Yaskawa INFORM job: X2_100(P)(125,-90).JBI

/JOB
//NAME X2_100(P)(125,-90)
//POS
///NPOS 391,391,391,27,0,0
///TOOL 0
///POSTYPE PULSE
///PULSE
C00000=15474,202180,164610,0,0,38
C00001=2027,202198,164679,0,0,38
C00002=24736,215365,219614,34446,41710,-28276
C00003=32352,212431,219590,43411,47182,-30672
C00004=90146,188560,202920,30112,59119,-18336
C00005=118933,140461,218744,27304,53624,2807
C00006=119754,138493,231524,24113,52403,6590
C00007=120507,123084,224138,21975,53379,9268
C00008=120855,115436,217153,22091,53699,9378
C00009=120999,112276,214168,22121,53888,9436
C00010=120994,108702,209954,21918,54592,9592
C00011=121002,109206,210530,21948,54503,9573
C00012=121014,109176,212154,22227,53559,9363
C00013=121002,109206,210530,21948,54503,9573
C00014=120510,120230,220891,21834,53874,9379
C00015=120545,123144,224216,-26507,40921,-26256
C00016=120895,115499,217236,-26128,41279,-26328
C00017=121036,110360,211926,-25743,41856,-26497
C00018=121034,108769,210044,-25582,42165,-26596
C00019=121035,109319,210673,-25631,42070,-26566
C00020=121049,109287,212294,-26118,41154,-26266
C00021=121035,109319,210673,-25631,42070,-26566
C00022=120543,120334,221019,-26244,41392,-26415
C00023=120983,122786,223558,-30476,46746,-26242
C00024=120987,115437,217242,-30421,46842,-26276
C00025=120987,110819,212678,-30218,47221,-26411
C00026=120984,108845,210344,-30028,47588,-26540
C00027=121056,109448,211035,-30038,47494,-26498
C00028=121070,109406,212645,-30499,46616,-26184
C00029=121056,109448,211035,-30038,47494,-26498
C00030=121048,120014,220398,-30195,47204,-26397
C00031=120925,149751,244690,-34380,46703,-25518
C00032=121565,167094,227706,-36094,61868,-28983
C00033=121107,161331,224195,-36551,61107,-28820
C00034=120919,157058,220850,-36681,60950,-28811
C00035=120917,155800,219633,-36648,61033,-28842
C00036=120923,156278,220067,-36652,61017,-28835
C00037=120930,157317,222816,-37031,60082,-28475
C00038=120923,156278,220067,-36652,61017,-28835
C00039=121567,164501,225300,-36048,61989,-29027
C00040=120589,166944,227359,-19824,59976,-30928
C00041=120819,161134,223823,-19888,59243,-30737
C00042=120912,157183,220866,-19892,59057,-30681
C00043=120909,155576,219240,-19859,59222,-30713
C00044=120921,156089,219731,-19862,59188,-30703
C00045=120928,157137,222490,-20094,58096,-30494
C00046=120921,156089,219731,-19862,59188,-30703
C00047=120597,164381,225001,-19795,60104,-30950
C00048=133714,167013,227584,29806,67145,20919
C00049=134110,161138,223906,30151,66407,20805
C00050=134262,157498,221144,30262,66227,20790
C00051=134252,155557,219269,30222,66366,20826
C00052=134278,156050,219725,30241,66337,20824
C00053=134486,157077,222435,30590,65306,20576
C00054=134278,156050,219725,30241,66337,20824
C00055=133722,164435,225200,29782,67268,20955
C00056=133985,188744,240463,29202,55916,39414
C00057=133788,188005,227705,27049,47808,60336
C00058=134139,183273,225821,27621,46590,60080
C00059=134274,179997,223870,27848,46130,59979
C00060=134264,178443,222562,27844,46137,59979
C00061=134276,178874,222921,27846,46135,59983
C00062=134459,180391,226047,28389,45077,59697
C00063=134276,178874,222921,27846,46135,59983
C00064=133784,185635,225817,27071,47759,60319
C00065=127585,202169,243145,858,47044,1942
C00066=121193,187855,227430,-25535,51149,-56270
C00067=120989,183220,225717,-26035,49903,-55992
C00068=120906,180048,223892,-26233,49429,-55882
C00069=120903,178425,222522,-26231,49435,-55886
C00070=120895,178865,222881,-26231,49438,-55890
C00071=120901,180413,226062,-26675,48393,-55581
C00072=120895,178865,222881,-26231,49438,-55890
C00073=121182,185490,225532,-25553,51104,-56261
C00074=121188,188192,227969,-25590,51004,-56232
C00075=120983,183552,226258,-26095,49755,-55951
C00076=120899,180084,224188,-26297,49279,-55843
C00077=120898,178760,223074,-26295,49283,-55844
C00078=120902,179187,223391,-26285,49306,-55850
C00079=120908,180723,226556,-26731,48265,-55540
C00080=120902,179187,223391,-26285,49306,-55850
C00081=121189,185816,226036,-25601,50976,-56224
C00082=123255,190499,236374,-58349,45147,30432
C00083=121547,184669,229695,-57916,45057,29536
C00084=120879,180825,225690,-57693,45050,29154
C00085=120877,179386,224486,-57692,45050,29153
C00086=120865,179866,224825,-57664,45066,29131
C00087=120860,178282,221599,-56698,45720,28507
C00088=120865,179866,224825,-57664,45066,29131
C00089=120725,179892,223679,-57103,45408,28721
C00090=120332,179896,223682,-57208,45243,28650
C00091=121348,179880,223660,-56933,45672,28832
C00092=123711,188247,233364,-57633,45714,30138
C00093=134983,214876,238244,-8707,44220,8832
C00094=134548,207430,231310,-8578,44619,8625
C00095=134367,202745,227274,-8541,44679,8550
C00096=134362,201870,226673,-8552,44600,8555
C00097=134379,202451,227139,-8553,44612,8561
C00098=134212,200435,223640,-8367,45704,8394
C00099=134379,202451,227139,-8553,44612,8561
C00100=134984,213013,237167,-8753,43928,8861
C00101=144264,210294,243886,-8163,41086,13861
C00102=162452,180370,234066,-6629,37835,23828
C00103=161533,173092,227071,-6569,38350,23478
C00104=162432,167522,220632,-6394,39487,23686
C00105=162432,166208,219497,-6392,39511,23685
C00106=162432,166481,219733,-6392,39506,23685
C00107=161891,165056,216873,-6255,40502,23429
C00108=162432,166481,219733,-6392,39506,23685
C00109=162497,178365,232600,-6647,37710,23854
C00110=147308,180890,237204,47154,21007,-10994
C00111=147638,173377,228129,43966,22135,-9369
C00112=147769,169207,223427,42684,22650,-8713
C00113=147776,167383,221906,42683,22648,-8711
C00114=147797,168129,222540,42691,22636,-8708
C00115=147426,166532,219395,41033,23590,-8010
C00116=147797,168129,222540,42691,22636,-8708
C00117=147340,178856,235656,47326,20933,-11067
C00118=133884,161941,227787,33603,50676,10210
C00119=127576,130559,218004,30921,63820,21625
C00120=128836,119462,220153,33793,57797,19920
C00121=129449,112387,214292,34197,57712,19962
C00122=129575,109480,211887,34296,57687,19970
C00123=132342,109409,211410,35968,57614,20273
C00124=135809,109300,210711,38054,57534,20678
C00125=138378,109197,210091,39570,57490,20998
C00126=138013,112115,212550,39343,57524,20963
C00127=137185,119214,218524,38825,57601,20885
C00128=115991,118707,218017,-25490,47827,-39243
C00129=116216,112084,213018,-25487,47549,-39133
C00130=116067,109362,210943,-25621,47425,-39117
C00131=124525,109336,210994,-20745,47997,-38204
C00132=124884,112043,212960,-20482,48190,-38202
C00133=124386,118675,218008,-20675,48440,-38320
C00134=123290,120759,219660,-35956,60120,-26268
C00135=122628,114303,214891,-36511,59734,-26205
C00136=121471,111489,212711,-37298,59521,-26266
C00137=122737,102232,205148,-46823,63858,-23746
C00138=124301,104933,207355,-45758,64087,-23652
C00139=125674,111471,212543,-44779,64387,-23617
C00140=122699,156385,234573,-36508,60394,-36922
C00141=122451,163606,222345,-33636,69881,-40152
C00142=121996,159570,221367,-34155,68543,-39836
C00143=121756,157914,220964,-34404,67985,-39712
C00144=120095,157879,220889,-35223,67629,-40000
C00145=118379,157761,220797,-36072,67224,-40285
C00146=122498,151785,218689,-44973,69197,-37741
C00147=123062,153607,219376,-44540,69722,-37837
C00148=123990,157704,220658,-43734,70938,-38144
C00149=117621,162254,221874,-19766,66589,-43069
C00150=117804,158098,220771,-19895,65240,-42790
C00151=117692,155503,219422,-20025,64751,-42727
C00152=123564,155493,219421,-17329,65494,-41580
C00153=123448,158048,220704,-17317,65981,-41679
C00154=123147,162227,221856,-17278,67320,-41949
C00155=130667,163848,224751,30344,74631,25358
C00156=131102,158990,222619,30735,73515,25150
C00157=131194,156955,221592,30843,73138,25067
C00158=136997,155740,218820,33776,72826,26305
C00159=136728,157787,219942,33579,73190,26353
C00160=136199,162650,222153,33133,74269,26558
C00161=131924,177838,230931,28709,51404,58848
C00162=131093,185219,225656,26178,57978,60553
C00163=131486,181652,225386,26742,56390,60255
C00164=131623,179818,224816,26950,55830,60146
C00165=136523,178332,222014,27857,55574,61608
C00166=136419,180039,222404,27637,56164,61742
C00167=135955,197166,232402,26774,58642,62268
C00168=123486,183195,222462,-21671,66302,-58170
C00169=123320,180439,223276,-22038,64485,-57858
C00170=123006,178865,223348,-22286,63635,-57774
C00171=118045,178731,223219,-23875,62688,-58963
C00172=118318,180513,223383,-23631,63488,-59060
C00173=118578,183298,222619,-23202,65292,-59373
C00174=122208,184099,222550,-27312,66798,-58279
C00175=121800,181437,223437,-27825,64995,-57938
C00176=121432,179848,223509,-28133,64143,-57821
C00177=118640,179803,223425,-29053,63504,-58468
C00178=122362,176158,223733,-39099,63902,-56258
C00179=122919,177928,223953,-38663,64680,-56393
C00180=123741,180697,223374,-37873,66345,-56772
C00181=125859,202099,241745,-26899,43318,-21165
C00182=128113,178960,235420,-24516,16567,13756
C00183=127689,171451,226207,-21929,18167,12428
C00184=127528,167831,221933,-20974,18864,11937
C00185=125917,168120,222387,-19991,18484,11020
C00186=112964,167943,221792,-9276,17273,2399
C00187=116391,165192,218668,-37133,21773,16827
C00188=116794,168607,222919,-38620,21196,17655
C00189=117426,176109,232276,-42123,19905,19505
C00190=121934,189549,236157,-2154,24440,9441
C00191=125766,180591,223933,31743,27648,1072
C00192=125872,172130,214005,30040,29143,1966
C00193=126601,167752,208377,28765,30022,2815
C00194=142051,161046,196707,20020,29981,11317
C00195=142147,165297,201916,20601,29000,11042
C00196=142364,174552,213002,21900,27026,10440
C00197=90146,188560,202920,30112,59119,-18336
C00198=32352,212431,219590,43411,47182,-30672
C00199=2027,202198,164679,0,0,38
C00200=15474,202180,164610,0,0,38
C00201=15474,202180,164610,0,0,38
C00202=15474,202180,164610,0,0,38
C00203=15474,202180,164610,0,0,38
C00204=15474,202180,164610,0,0,38
C00205=-58614,195716,224396,-17895,28031,-14924
C00206=-117113,152285,229609,-38431,39797,-17389
C00207=-135921,136983,237719,-46639,40267,-16819
C00208=-146165,113701,216007,-48123,45886,-19082
C00209=-147115,109767,211721,-48018,46725,-19481
C00210=-147088,107791,209384,-47709,47018,-19672
C00211=-147094,108297,209962,-47779,46951,-19629
C00212=-147691,108253,211472,-48816,46225,-19236
C00213=-147094,108297,209962,-47779,46951,-19629
C00214=-145940,119401,220708,-47691,46482,-19124
C00215=-145956,122257,223946,12736,42114,23473
C00216=-146776,114562,216701,12165,42638,23451
C00217=-149521,110157,218004,11318,39720,22735
C00218=-147064,107789,209368,11782,43659,23556
C00219=-152611,108638,222377,10271,36372,22002
C00220=-147661,108297,211513,11684,42643,23344
C00221=-152611,108638,222377,10271,36372,22002
C00222=-145911,119443,220742,12635,42626,23555
C00223=-129100,127332,227576,23440,42260,25369
C00224=-99845,140323,234668,41114,43975,29200
C00225=-81288,119441,205391,47500,48209,34399
C00226=-80509,111680,198241,47632,48326,34680
C00227=-79929,105264,191953,47555,48593,35008
C00228=-79929,103140,189447,47268,48904,35206
C00229=-79929,103522,189901,47320,48847,35170
C00230=-79411,103879,191333,48035,48251,34928
C00231=-80657,107851,193513,46953,49010,35078
C00232=-81393,116289,201791,47062,48643,34649
C00233=-121441,148548,228494,40235,53726,25728
C00234=-121126,165586,226218,36457,61785,29251
C00235=-120656,159787,222623,36910,61050,29098
C00236=-120465,155988,219703,37047,60878,29083
C00237=-120464,154211,217972,36998,61001,29130
C00238=-120470,154693,218414,37003,60983,29122
C00239=-120461,155760,221201,37395,60041,28759
C00240=-120470,154693,218414,37003,60983,29122
C00241=-121130,162973,223775,36406,61917,29299
C00242=-120157,165759,226450,20196,59859,31167
C00243=-120376,159925,222865,20264,59145,30979
C00244=-120465,156088,219927,20262,59004,30931
C00245=-120464,154338,218223,20232,59143,30959
C00246=-120475,154854,218720,20235,59107,30949
C00247=-120466,155913,221497,20480,58011,30738
C00248=-120475,154854,218720,20235,59107,30949
C00249=-120168,163183,224065,20164,59996,31190
C00250=-146488,166005,227001,-35633,64430,-23031
C00251=-147030,160017,223073,-36069,63762,-22930
C00252=-147236,156149,220027,-36198,63621,-22931
C00253=-147219,154376,218307,-36149,63745,-22972
C00254=-147245,154867,218758,-36168,63719,-22970
C00255=-147633,155852,221361,-36670,62738,-22707
C00256=-147245,154867,218758,-36168,63719,-22970
C00257=-146483,163417,224595,-35590,64555,-23074
C00258=-120317,171933,242187,-34338,35763,-50845
C00259=-120155,165766,226473,-29925,41593,-53256
C00260=-120374,159929,222883,-30422,40861,-53041
C00261=-120463,156296,220142,-30547,40687,-53000
C00262=-120462,154340,218238,-30449,40831,-53058
C00263=-120473,154616,218516,-30468,40803,-53050
C00264=-120468,155465,220597,-30969,40075,-52744
C00265=-120473,154822,218708,-30475,40793,-53046
C00266=-120165,163158,224064,-29848,41715,-53306
C00267=-120812,165753,226464,30411,41431,53453
C00268=-120571,159914,222865,30920,40700,53240
C00269=-120472,156279,220119,31048,40527,53200
C00270=-120471,154323,218216,30948,40670,53260
C00271=-120462,154817,218686,30971,40637,53250
C00272=-120453,155874,221461,31687,39633,52832
C00273=-120462,154817,218686,30971,40637,53250
C00274=-120802,163155,224052,30328,41558,53507
C00275=-120794,196445,225743,23944,55971,57861
C00276=-120590,192435,224899,24399,54512,57575
C00277=-120507,189535,223519,24597,53909,57452
C00278=-120506,188039,222351,24612,53862,57441
C00279=-120510,188436,222616,24600,53901,57449
C00280=-120503,190244,226011,24956,52841,57180
C00281=-120510,188436,222616,24600,53901,57449
C00282=-120797,194186,224030,23972,55873,57836
C00283=-120994,201212,234683,5149,48132,-3005
C00284=-136826,197795,228776,4624,50735,-8156
C00285=-136826,191727,224657,4661,50153,-8183
C00286=-138745,198654,246113,16555,26136,-13965
C00287=-138745,196808,244858,16658,25967,-14016
C00288=-138745,198654,246113,16555,26136,-13965
C00289=-138556,197554,243943,16057,26850,-13661
C00290=-138745,198654,246113,16555,26136,-13965
C00291=-120778,201953,235347,5155,48094,-2935
C00292=-122925,194375,228384,5084,48585,-3628
C00293=-122022,191255,226196,5106,48287,-3341
C00294=-122022,188924,224535,5119,48113,-3349
C00295=-122022,191255,226196,5106,48287,-3341
C00296=-122007,189355,222871,5025,49352,-3280
C00297=-122022,191255,226196,5106,48287,-3341
C00298=-120785,199939,233992,5171,47894,-2948
C00299=-121100,206663,244168,5684,44070,-5780
C00300=-121083,191157,235435,5956,40419,-9249
C00301=-120661,183492,227908,5865,41088,-9055
C00302=-120495,180342,224726,5822,41418,-8974
C00303=-120493,177643,222664,5836,41300,-8982
C00304=-120497,178404,223351,5840,41268,-8985
C00305=-120504,176471,219821,5709,42442,-8908
C00306=-120497,178404,223351,5840,41268,-8985
C00307=-121086,189297,234244,5983,40198,-9266
C00308=-146820,179847,236540,-47569,21348,11498
C00309=-147178,172319,227421,-44381,22472,9861
C00310=-147319,168316,222840,-43092,22988,9195
C00311=-147327,166302,221149,-43081,22990,9188
C00312=-147348,167051,221792,-43093,22976,9188
C00313=-146991,165439,218615,-41422,23930,8479
C00314=-147348,167051,221792,-43093,22976,9188
C00315=-146852,177807,234978,-47728,21278,11565
C00316=-135233,175637,232065,-30395,22918,7865
C00317=-134932,170558,225163,-28644,24419,7102
C00318=-134048,167164,221268,-28229,25184,7160
C00319=-151719,157645,202807,-16034,27960,-3795
C00320=-149884,166658,215825,-18859,24998,-1880
C00321=-146998,184619,240811,-25863,19770,2323
C00322=-125978,166364,224291,9417,26840,-6325
C00323=-129674,155803,216839,10617,26282,-8064
C00324=-129498,149917,208752,9902,28190,-7650
C00325=-128727,145711,203487,9397,29196,-7156
C00326=-146983,136453,186134,10957,36521,-13611
C00327=-147815,150895,204985,12306,32503,-14599
C00328=-147815,166494,219236,12563,31767,-14734
C00329=-117911,183214,223223,-22567,61413,-57159
C00330=-118075,179761,223119,-22973,59798,-56859
C00331=-118640,177544,221909,-23214,59324,-56920
C00332=-123472,177522,221869,-24524,58369,-58124
C00333=-123089,179795,223206,-24339,58762,-58103
C00334=-122842,183276,223359,-23878,60366,-58401
C00335=-123442,190112,227842,21784,66477,58404
C00336=-123264,179517,222829,22229,64249,58012
C00337=-123470,177948,222872,22311,63517,57806
C00338=-118464,178077,223118,23939,62475,58981
C00339=-118255,179504,222781,23818,63292,59223
C00340=-118526,182312,222057,23382,65085,59534
C00341=-122160,182951,221704,27481,66647,58451
C00342=-121741,180270,222553,28000,64855,58113
C00343=-121841,178346,222179,28131,64207,57913
C00344=-118577,178303,222154,29213,63422,58659
C00345=-122472,175017,222795,39229,63796,56395
C00346=-122854,176802,223069,38864,64502,56556
C00347=-123688,179595,222537,38068,66154,56931
C00348=-122762,177463,230138,35132,68647,45006
C00349=-122410,162609,221657,33920,69712,40281
C00350=-121942,158550,220632,34447,68388,39967
C00351=-122084,156654,219964,34496,67953,39787
C00352=-118316,156835,220042,36358,67113,40432
C00353=-122608,150908,218064,45207,69057,37831
C00354=-122995,152587,218620,44867,69536,37955
C00355=-123937,156712,219961,44053,70736,38256
C00356=-117567,161316,221321,20040,66440,43208
C00357=-117737,157140,220183,20178,65102,42929
C00358=-118356,154594,218971,19982,64654,42713
C00359=-123958,154557,218888,17402,65396,41629
C00360=-123397,157158,220257,17595,65803,41812
C00361=-123107,161358,221443,17548,67132,42081
C00362=-143812,163767,225728,-37102,71366,-27286
C00363=-144478,158774,223325,-37668,70333,-27076
C00364=-145574,156483,221747,-38290,69906,-27183
C00365=-150790,154198,216554,-40571,70164,-28612
C00366=-149872,156514,218237,-40068,70526,-28516
C00367=-149135,161509,220758,-39481,71513,-28708
C00368=-132073,148583,237547,-34621,60846,-21391
C00369=-128841,120799,222047,-33572,57550,-19735
C00370=-130509,111569,213679,-34507,57728,-19991
C00371=-142163,108136,208271,-41379,57632,-21462
C00372=-150058,107393,204742,-45605,57822,-22784
C00373=-138074,111342,212170,-39066,57558,-20867
C00374=-137251,118465,218184,-38555,57622,-20786
C00375=-115920,117937,217688,25888,47668,39306
C00376=-117242,111297,212709,25258,47458,39075
C00377=-117220,108280,210223,25280,47439,39073
C00378=-125843,108493,210262,20260,48127,38171
C00379=-124861,111270,212684,20846,48005,38264
C00380=-124377,117927,217775,21034,48243,38378
C00381=-123273,119993,219247,36349,59987,26322
C00382=-122589,113511,214424,36914,59617,26265
C00383=-122996,110841,212352,36684,59583,26203
C00384=-117053,110850,212325,40539,58921,26676
C00385=-124086,101367,204591,46303,63921,23704
C00386=-124243,104084,206817,46189,63960,23705
C00387=-125643,110657,212075,45198,64245,23661
C00388=-113480,133194,224663,34991,55578,15993
C00389=-58614,195716,224396,-17895,28031,-14924
C00390=15474,202180,164610,0,0,38
BC00000=0,675528,1075229
BC00001=0,1249520,1075229
BC00002=20074,1273230,1075229
BC00003=22843,1276500,1075229
BC00004=181219,1349640,881743
BC00005=259614,1271622,997019
BC00006=263455,1253369,961473
BC00007=265649,1242939,941161
BC00008=265649,1242939,941161
BC00009=265649,1242939,941161
BC00010=265649,1242939,941161
BC00011=265649,1242939,941161
BC00012=265649,1242939,941161
BC00013=265649,1242939,941161
BC00014=265649,1242939,941161
BC00015=279094,1259762,979345
BC00016=279094,1259762,979345
BC00017=279094,1259762,979345
BC00018=279094,1259762,979345
BC00019=279094,1259762,979345
BC00020=279094,1259762,979345
BC00021=279094,1259762,979345
BC00022=279094,1259762,979345
BC00023=338482,1253298,958814
BC00024=338482,1253298,958814
BC00025=338482,1253298,958814
BC00026=338482,1253298,958814
BC00027=338482,1253298,958814
BC00028=338482,1253298,958814
BC00029=338482,1253298,958814
BC00030=338482,1253298,958814
BC00031=333821,1266832,919202
BC00032=321005,1304050,810268
BC00033=321005,1304050,810268
BC00034=321005,1304050,810268
BC00035=321005,1304050,810268
BC00036=321005,1304050,810268
BC00037=321005,1304050,810268
BC00038=321005,1304050,810268
BC00039=321005,1304050,810268
BC00040=279090,1297669,836196
BC00041=279090,1297669,836196
BC00042=279090,1297669,836196
BC00043=279090,1297669,836196
BC00044=279090,1297669,836196
BC00045=279090,1297669,836196
BC00046=279090,1297669,836196
BC00047=279090,1297669,836196
BC00048=308990,1283728,803935
BC00049=308990,1283728,803935
BC00050=308990,1283728,803935
BC00051=308990,1283728,803935
BC00052=308990,1283728,803935
BC00053=308990,1283728,803935
BC00054=308990,1283728,803935
BC00055=308990,1283728,803935
BC00056=309388,1296619,799441
BC00057=309813,1310369,794648
BC00058=309813,1310369,794648
BC00059=309813,1310369,794648
BC00060=309813,1310369,794648
BC00061=309813,1310369,794648
BC00062=309813,1310369,794648
BC00063=309813,1310369,794648
BC00064=309813,1310369,794648
BC00065=290509,1311906,794287
BC00066=271204,1313444,793926
BC00067=271204,1313444,793926
BC00068=271204,1313444,793925
BC00069=271204,1313444,793926
BC00070=271204,1313444,793926
BC00071=271204,1313444,793926
BC00072=271204,1313444,793926
BC00073=271204,1313444,793926
BC00074=339752,1313535,794120
BC00075=339752,1313535,794120
BC00076=339752,1313535,794120
BC00077=339752,1313535,794120
BC00078=339752,1313535,794120
BC00079=339752,1313535,794120
BC00080=339752,1313535,794120
BC00081=339752,1313535,794120
BC00082=309596,1336055,723788
BC00083=309596,1336055,723788
BC00084=309596,1336055,723788
BC00085=309596,1336055,723788
BC00086=309596,1336055,723788
BC00087=309596,1336055,723788
BC00088=309596,1336055,723788
BC00089=309596,1336055,723788
BC00090=309596,1336055,723788
BC00091=309596,1336055,723788
BC00092=309596,1336055,723788
BC00093=366840,1349942,659049
BC00094=366840,1349942,659049
BC00095=366840,1349942,659049
BC00096=366840,1349942,659049
BC00097=366840,1349942,659049
BC00098=366840,1349942,659049
BC00099=366840,1349942,659049
BC00100=366840,1349942,659049
BC00101=369598,1321086,746352
BC00102=375224,1262220,924452
BC00103=375224,1262220,924452
BC00104=375224,1262220,924452
BC00105=375224,1262220,924452
BC00106=375224,1262220,924452
BC00107=375224,1262220,924450
BC00108=375224,1262220,924452
BC00109=375224,1262220,924452
BC00110=339925,1300732,881743
BC00111=339925,1300732,881743
BC00112=339925,1300732,881743
BC00113=339925,1300732,881743
BC00114=339925,1300732,881743
BC00115=339925,1300732,881743
BC00116=339925,1300732,881743
BC00117=339925,1300732,881743
BC00118=315652,1292340,901479
BC00119=299654,1262212,953023
BC00120=298993,1238691,912276
BC00121=298993,1238691,912276
BC00122=298993,1238691,912274
BC00123=298993,1238691,912276
BC00124=298993,1238691,912276
BC00125=298993,1238691,912276
BC00126=298993,1238691,912276
BC00127=298993,1238691,912276
BC00128=278815,1248832,951478
BC00129=278815,1248832,951478
BC00130=278815,1248832,951478
BC00131=278815,1248832,951478
BC00132=278815,1248832,951478
BC00133=278815,1248832,951478
BC00134=314804,1246682,892728
BC00135=314804,1246682,892728
BC00136=314804,1246682,892728
BC00137=314804,1246682,892728
BC00138=314804,1246682,892728
BC00139=314804,1246682,892728
BC00140=314801,1292959,892910
BC00141=314719,1294052,772836
BC00142=314719,1294052,772836
BC00143=314719,1294052,772836
BC00144=314719,1294052,772836
BC00145=314719,1294052,772836
BC00146=314719,1294052,772836
BC00147=314719,1294052,772836
BC00148=314719,1294052,772836
BC00149=278878,1286739,810029
BC00150=278878,1286739,810029
BC00151=278878,1286739,810029
BC00152=278878,1286739,810029
BC00153=278878,1286739,810029
BC00154=278878,1286739,810029
BC00155=311908,1275469,768683
BC00156=311908,1275469,768683
BC00157=311908,1275469,768683
BC00158=311908,1275469,768683
BC00159=311908,1275469,768683
BC00160=311908,1275469,768683
BC00161=311248,1293583,920117
BC00162=310634,1294320,778613
BC00163=310634,1294320,778613
BC00164=310635,1294320,778611
BC00165=310635,1294320,778611
BC00166=310634,1294320,778613
BC00167=310634,1294320,778613
BC00168=269571,1288878,766650
BC00169=269571,1288878,766650
BC00170=269571,1288878,766650
BC00171=269571,1288878,766650
BC00172=269571,1288878,766650
BC00173=269571,1288878,766650
BC00174=324029,1292263,751538
BC00175=324029,1292263,751538
BC00176=324029,1292263,751538
BC00177=324029,1292263,751538
BC00178=324029,1292263,751538
BC00179=324029,1292263,751538
BC00180=324029,1292263,751538
BC00181=331457,1324273,767907
BC00182=337552,1339765,848258
BC00183=337552,1339765,848258
BC00184=337551,1339764,848257
BC00185=337552,1339765,848258
BC00186=337552,1339765,848258
BC00187=337552,1339765,848258
BC00188=337552,1339765,848258
BC00189=337552,1339765,848258
BC00190=326395,1340304,844891
BC00191=315775,1339017,839253
BC00192=315775,1339017,839253
BC00193=315775,1339017,839253
BC00194=315775,1339017,839253
BC00195=315775,1339017,839253
BC00196=315775,1339017,839253
BC00197=181219,1349640,881743
BC00198=22843,1276500,1075229
BC00199=0,1249520,1075229
BC00200=0,675528,1075229
BC00201=0,675528,1075229
BC00202=0,675528,1075229
BC00203=0,675528,1075229
BC00204=0,675528,1075229
BC00205=138607,763027,1056836
BC00206=261748,840763,986656
BC00207=303122,866882,963076
BC00208=320914,878114,952936
BC00209=322510,879121,952026
BC00210=322510,879121,952026
BC00211=322510,879121,952026
BC00212=322510,879121,952026
BC00213=322510,879121,952026
BC00214=322510,879121,952026
BC00215=326477,871688,980713
BC00216=326477,871688,980713
BC00217=326477,883252,980713
BC00218=326477,871688,980713
BC00219=326477,895644,980713
BC00220=326477,871688,980713
BC00221=326477,895644,980713
BC00222=326477,871688,980713
BC00223=304746,865718,972507
BC00224=267497,855485,958441
BC00225=255081,864777,953752
BC00226=255081,864777,953752
BC00227=255081,864777,953752
BC00228=255081,864777,953752
BC00229=255081,864777,953752
BC00230=255081,864777,953752
BC00231=255081,864777,953752
BC00232=255081,864777,953752
BC00233=320924,819371,961652
BC00234=320924,819371,812233
BC00235=320924,819371,812233
BC00236=320924,819371,812233
BC00237=320924,819371,812233
BC00238=320924,819371,812233
BC00239=320924,819371,812233
BC00240=320924,819371,812233
BC00241=320924,819371,812233
BC00242=278908,825639,838037
BC00243=278908,825639,838037
BC00244=278908,825639,838037
BC00245=278908,825639,838037
BC00246=278908,825639,838037
BC00247=278908,825639,838037
BC00248=278908,825639,838037
BC00249=278908,825639,838037
BC00250=344258,850073,804397
BC00251=344258,850073,804397
BC00252=344258,850073,804397
BC00253=344258,850073,804397
BC00254=344258,850073,804397
BC00255=344258,850073,804397
BC00256=344258,850073,804397
BC00257=344258,850073,804397
BC00258=268540,837164,928608
BC00259=268540,837164,928608
BC00260=268540,837164,928608
BC00261=268540,837164,928608
BC00262=268540,837164,928608
BC00263=268540,837164,928608
BC00264=268541,837164,928607
BC00265=268540,837164,928608
BC00266=268540,837164,928608
BC00267=271645,836699,929417
BC00268=271645,836699,929417
BC00269=271645,836699,929417
BC00270=271645,836699,929417
BC00271=271645,836699,929417
BC00272=271645,836699,929417
BC00273=271645,836699,929417
BC00274=271645,836699,929417
BC00275=340192,799254,723936
BC00276=340192,799254,723936
BC00277=340192,799254,723936
BC00278=340192,799254,723936
BC00279=340192,799254,723936
BC00280=340192,799254,723936
BC00281=340192,799254,723936
BC00282=340192,799254,723936
BC00283=321646,797982,745635
BC00284=321646,797982,745635
BC00285=321646,797982,745635
BC00286=321646,797982,745635
BC00287=321646,797982,745635
BC00288=321646,797982,745635
BC00289=321646,797982,745635
BC00290=321646,797982,745635
BC00291=321646,797982,745635
BC00292=321646,797982,745635
BC00293=321646,797984,745632
BC00294=321646,797984,745632
BC00295=321646,797984,745632
BC00296=321646,797984,745632
BC00297=321646,797984,745632
BC00298=321646,797982,745635
BC00299=296475,807012,791430
BC00300=260705,819844,856508
BC00301=260705,819844,856508
BC00302=260705,819844,856508
BC00303=260705,819844,856508
BC00304=260705,819844,856508
BC00305=260705,819844,856508
BC00306=260705,819844,856508
BC00307=260705,819844,856508
BC00308=339123,823007,883432
BC00309=339123,823007,883432
BC00310=339123,823007,883432
BC00311=339123,823007,883432
BC00312=339123,823007,883432
BC00313=339123,823007,883432
BC00314=339123,823007,883432
BC00315=339123,823007,883432
BC00316=339668,815369,895136
BC00317=339668,815369,895136
BC00318=339668,815369,895136
BC00319=339682,815172,895438
BC00320=339682,815172,895438
BC00321=339682,815172,895438
BC00322=343473,807454,949850
BC00323=343473,807454,949850
BC00324=343473,807454,949850
BC00325=343471,807456,949849
BC00326=343517,807585,950150
BC00327=343517,807585,950150
BC00328=343517,807585,950150
BC00329=270260,826762,778340
BC00330=270260,826762,778340
BC00331=270260,826762,778339
BC00332=270260,826762,778339
BC00333=270260,826762,778340
BC00334=270260,826762,778340
BC00335=270830,834917,768745
BC00336=270830,834917,768745
BC00337=270830,834917,768745
BC00338=270830,834917,768745
BC00339=270830,834917,768745
BC00340=270830,834917,768745
BC00341=325301,832050,753660
BC00342=325301,832050,753660
BC00343=325301,832050,753660
BC00344=325301,832050,753660
BC00345=325301,832050,753660
BC00346=325301,832050,753660
BC00347=325301,832050,753660
BC00348=317689,831131,771467
BC00349=315834,830096,774743
BC00350=315834,830096,774743
BC00351=315834,830096,774743
BC00352=315834,830096,774743
BC00353=315834,830096,774743
BC00354=315834,830096,774743
BC00355=315834,830096,774743
BC00356=279937,837039,812006
BC00357=279937,837039,812006
BC00358=279937,837039,812006
BC00359=279937,837039,812006
BC00360=279937,837039,812006
BC00361=279937,837039,812006
BC00362=348145,858726,767388
BC00363=348145,858726,767388
BC00364=348145,858726,767388
BC00365=348145,858726,767388
BC00366=348145,858726,767388
BC00367=348145,858726,767388
BC00368=304168,872987,860177
BC00369=299744,886342,911434
BC00370=299744,886342,911434
BC00371=320499,886342,911434
BC00372=320499,886342,911434
BC00373=299744,886342,911434
BC00374=299744,886342,911434
BC00375=280164,875026,952983
BC00376=280164,875026,952983
BC00377=280164,875026,952983
BC00378=280164,875026,952983
BC00379=280164,875026,952983
BC00380=280164,875026,952983
BC00381=315859,877538,894138
BC00382=315859,877538,894138
BC00383=315859,877538,894138
BC00384=315859,877538,894138
BC00385=315859,877538,894138
BC00386=315859,877538,894138
BC00387=315859,877538,894138
BC00388=284199,857085,923198
BC00389=138607,763027,1056836
BC00390=0,675528,1075229
EC00000=1108551,-556475
EC00001=1108551,-556475
EC00002=1108551,-556475
EC00003=1108551,-556475
EC00004=1108551,-556475
EC00005=1108551,-556475
EC00006=1108551,-556475
EC00007=1108551,-556475
EC00008=1108551,-556475
EC00009=1108551,-556475
EC00010=1108551,-556475
EC00011=1108551,-556475
EC00012=1108551,-556475
EC00013=1108551,-556475
EC00014=1108551,-556475
EC00015=1108551,-556475
EC00016=1108551,-556475
EC00017=1108551,-556475
EC00018=1108551,-556475
EC00019=1108551,-556475
EC00020=1108551,-556475
EC00021=1108551,-556475
EC00022=1108551,-556475
EC00023=1108551,-556475
EC00024=1108551,-556475
EC00025=1108551,-556475
EC00026=1108551,-556475
EC00027=1108551,-556475
EC00028=1108551,-556475
EC00029=1108551,-556475
EC00030=1108551,-556475
EC00031=1108551,-556475
EC00032=1108551,-556475
EC00033=1108551,-556475
EC00034=1108551,-556475
EC00035=1108551,-556475
EC00036=1108551,-556475
EC00037=1108551,-556475
EC00038=1108551,-556475
EC00039=1108551,-556475
EC00040=1108551,-556475
EC00041=1108551,-556475
EC00042=1108551,-556475
EC00043=1108551,-556475
EC00044=1108551,-556475
EC00045=1108551,-556475
EC00046=1108551,-556475
EC00047=1108551,-556475
EC00048=1108551,-556475
EC00049=1108551,-556475
EC00050=1108551,-556475
EC00051=1108551,-556475
EC00052=1108551,-556475
EC00053=1108551,-556475
EC00054=1108551,-556475
EC00055=1108551,-556475
EC00056=1108551,-556475
EC00057=1108551,-556475
EC00058=1108551,-556475
EC00059=1108551,-556475
EC00060=1108551,-556475
EC00061=1108551,-556475
EC00062=1108551,-556475
EC00063=1108551,-556475
EC00064=1108551,-556475
EC00065=1108551,-556475
EC00066=1108551,-556475
EC00067=1108551,-556475
EC00068=1108550,-556475
EC00069=1108551,-556475
EC00070=1108551,-556475
EC00071=1108551,-556475
EC00072=1108551,-556475
EC00073=1108551,-556475
EC00074=1108551,-556475
EC00075=1108551,-556475
EC00076=1108551,-556475
EC00077=1108551,-556475
EC00078=1108551,-556475
EC00079=1108551,-556475
EC00080=1108551,-556475
EC00081=1108551,-556475
EC00082=1108551,-556475
EC00083=1108551,-556475
EC00084=1108551,-556475
EC00085=1108551,-556475
EC00086=1108551,-556475
EC00087=1108551,-556475
EC00088=1108551,-556475
EC00089=1108551,-556475
EC00090=1108551,-556475
EC00091=1108551,-556475
EC00092=1108551,-556475
EC00093=1108551,-556475
EC00094=1108551,-556475
EC00095=1108551,-556475
EC00096=1108551,-556475
EC00097=1108551,-556475
EC00098=1108551,-556475
EC00099=1108551,-556475
EC00100=1108551,-556475
EC00101=1108551,-556475
EC00102=1108551,-556475
EC00103=1108551,-556475
EC00104=1108551,-556475
EC00105=1108551,-556475
EC00106=1108551,-556475
EC00107=1108550,-556474
EC00108=1108551,-556475
EC00109=1108551,-556475
EC00110=1108551,-556475
EC00111=1108551,-556475
EC00112=1108551,-556475
EC00113=1108551,-556475
EC00114=1108551,-556475
EC00115=1108551,-556475
EC00116=1108551,-556475
EC00117=1108551,-556475
EC00118=1108551,-556475
EC00119=1108551,-556475
EC00120=1108551,-556475
EC00121=1108551,-556475
EC00122=1108551,-556474
EC00123=1108551,-556475
EC00124=1108551,-556475
EC00125=1108551,-556475
EC00126=1108551,-556475
EC00127=1108551,-556475
EC00128=1108551,-556475
EC00129=1108551,-556475
EC00130=1108551,-556475
EC00131=1108551,-556475
EC00132=1108551,-556475
EC00133=1108551,-556475
EC00134=1108551,-556475
EC00135=1108551,-556475
EC00136=1108551,-556475
EC00137=1108551,-556475
EC00138=1108551,-556475
EC00139=1108551,-556475
EC00140=1108551,-556475
EC00141=1108551,-556475
EC00142=1108551,-556475
EC00143=1108551,-556475
EC00144=1108551,-556475
EC00145=1108551,-556475
EC00146=1108551,-556475
EC00147=1108551,-556475
EC00148=1108551,-556475
EC00149=1108551,-556475
EC00150=1108551,-556475
EC00151=1108551,-556475
EC00152=1108551,-556475
EC00153=1108551,-556475
EC00154=1108551,-556475
EC00155=1108551,-556475
EC00156=1108551,-556475
EC00157=1108551,-556475
EC00158=1108551,-556475
EC00159=1108551,-556475
EC00160=1108551,-556475
EC00161=1108551,-556475
EC00162=1108551,-556475
EC00163=1108551,-556475
EC00164=1108550,-556475
EC00165=1108550,-556475
EC00166=1108551,-556475
EC00167=1108551,-556475
EC00168=1108551,-556475
EC00169=1108551,-556475
EC00170=1108551,-556475
EC00171=1108551,-556475
EC00172=1108551,-556475
EC00173=1108551,-556475
EC00174=1108551,-556475
EC00175=1108551,-556475
EC00176=1108551,-556475
EC00177=1108551,-556475
EC00178=1108551,-556475
EC00179=1108551,-556475
EC00180=1108551,-556475
EC00181=1108551,-556475
EC00182=1108551,-556475
EC00183=1108551,-556475
EC00184=1108550,-556475
EC00185=1108551,-556475
EC00186=1108551,-556475
EC00187=1108551,-556475
EC00188=1108551,-556475
EC00189=1108551,-556475
EC00190=1108551,-556475
EC00191=1108551,-556475
EC00192=1108551,-556475
EC00193=1108551,-556475
EC00194=1108551,-556475
EC00195=1108551,-556475
EC00196=1108551,-556475
EC00197=1108551,-556475
EC00198=1108551,-556475
EC00199=1108551,-556475
EC00200=1108551,-556475
EC00201=1108551,-556475
EC00202=266052,-556475
EC00203=-266052,556475
EC00204=-1108551,556475
EC00205=-1108551,556475
EC00206=-1108551,556475
EC00207=-1108551,556475
EC00208=-1108551,556475
EC00209=-1108551,556475
EC00210=-1108551,556475
EC00211=-1108551,556475
EC00212=-1108551,556475
EC00213=-1108551,556475
EC00214=-1108551,556475
EC00215=-1108551,556475
EC00216=-1108551,556475
EC00217=-1108551,556475
EC00218=-1108551,556475
EC00219=-1108551,556475
EC00220=-1108551,556475
EC00221=-1108551,556475
EC00222=-1108551,556475
EC00223=-1108551,556475
EC00224=-1108551,556475
EC00225=-1108551,556475
EC00226=-1108551,556475
EC00227=-1108551,556475
EC00228=-1108551,556475
EC00229=-1108551,556475
EC00230=-1108551,556475
EC00231=-1108551,556475
EC00232=-1108551,556475
EC00233=-1108551,556475
EC00234=-1108551,556475
EC00235=-1108551,556475
EC00236=-1108551,556475
EC00237=-1108551,556475
EC00238=-1108551,556475
EC00239=-1108551,556475
EC00240=-1108551,556475
EC00241=-1108551,556475
EC00242=-1108551,556475
EC00243=-1108551,556475
EC00244=-1108551,556475
EC00245=-1108551,556475
EC00246=-1108551,556475
EC00247=-1108551,556475
EC00248=-1108551,556475
EC00249=-1108551,556475
EC00250=-1108551,556475
EC00251=-1108551,556475
EC00252=-1108551,556475
EC00253=-1108551,556475
EC00254=-1108551,556475
EC00255=-1108551,556475
EC00256=-1108551,556475
EC00257=-1108551,556475
EC00258=-1108551,556475
EC00259=-1108551,556475
EC00260=-1108551,556475
EC00261=-1108551,556475
EC00262=-1108551,556475
EC00263=-1108551,556475
EC00264=-1108550,556475
EC00265=-1108551,556475
EC00266=-1108551,556475
EC00267=-1108551,556475
EC00268=-1108551,556475
EC00269=-1108551,556475
EC00270=-1108551,556475
EC00271=-1108551,556475
EC00272=-1108551,556475
EC00273=-1108551,556475
EC00274=-1108551,556475
EC00275=-1108551,556475
EC00276=-1108551,556475
EC00277=-1108551,556475
EC00278=-1108551,556475
EC00279=-1108551,556475
EC00280=-1108551,556475
EC00281=-1108551,556475
EC00282=-1108551,556475
EC00283=-1108551,556475
EC00284=-1108551,556475
EC00285=-1108551,556475
EC00286=-1108551,556475
EC00287=-1108551,556475
EC00288=-1108551,556475
EC00289=-1108551,556475
EC00290=-1108551,556475
EC00291=-1108551,556475
EC00292=-1108551,556475
EC00293=-1108550,556475
EC00294=-1108550,556475
EC00295=-1108550,556475
EC00296=-1108550,556475
EC00297=-1108550,556475
EC00298=-1108551,556475
EC00299=-1108551,556475
EC00300=-1108551,556475
EC00301=-1108551,556475
EC00302=-1108551,556475
EC00303=-1108551,556475
EC00304=-1108551,556475
EC00305=-1108551,556475
EC00306=-1108551,556475
EC00307=-1108551,556475
EC00308=-1108551,556475
EC00309=-1108551,556475
EC00310=-1108551,556475
EC00311=-1108551,556475
EC00312=-1108551,556475
EC00313=-1108551,556475
EC00314=-1108551,556475
EC00315=-1108551,556475
EC00316=-1108549,556476
EC00317=-1108549,556476
EC00318=-1108549,556476
EC00319=-1108549,556476
EC00320=-1108549,556476
EC00321=-1108549,556476
EC00322=-1108551,556475
EC00323=-1108551,556475
EC00324=-1108551,556475
EC00325=-1108551,556476
EC00326=-1108551,556475
EC00327=-1108551,556475
EC00328=-1108551,556475
EC00329=-1108551,556475
EC00330=-1108551,556475
EC00331=-1108550,556476
EC00332=-1108550,556476
EC00333=-1108551,556475
EC00334=-1108551,556475
EC00335=-1108551,556475
EC00336=-1108551,556475
EC00337=-1108551,556475
EC00338=-1108551,556475
EC00339=-1108551,556475
EC00340=-1108551,556475
EC00341=-1108551,556475
EC00342=-1108551,556475
EC00343=-1108551,556475
EC00344=-1108551,556475
EC00345=-1108551,556475
EC00346=-1108551,556475
EC00347=-1108551,556475
EC00348=-1108551,556475
EC00349=-1108551,556475
EC00350=-1108551,556475
EC00351=-1108551,556475
EC00352=-1108551,556475
EC00353=-1108551,556475
EC00354=-1108551,556475
EC00355=-1108551,556475
EC00356=-1108551,556475
EC00357=-1108551,556475
EC00358=-1108551,556475
EC00359=-1108551,556475
EC00360=-1108551,556475
EC00361=-1108551,556475
EC00362=-1108551,556475
EC00363=-1108551,556475
EC00364=-1108551,556475
EC00365=-1108551,556475
EC00366=-1108551,556475
EC00367=-1108551,556475
EC00368=-1108551,556475
EC00369=-1108551,556475
EC00370=-1108551,556475
EC00371=-1108551,556475
EC00372=-1108551,556475
EC00373=-1108551,556475
EC00374=-1108551,556475
EC00375=-1108551,556475
EC00376=-1108551,556475
EC00377=-1108551,556475
EC00378=-1108551,556475
EC00379=-1108551,556475
EC00380=-1108551,556475
EC00381=-1108551,556475
EC00382=-1108551,556475
EC00383=-1108551,556475
EC00384=-1108551,556475
EC00385=-1108551,556475
EC00386=-1108551,556475
EC00387=-1108551,556475
EC00388=-1108551,556475
EC00389=-1108551,556475
EC00390=-1108551,556475
///POSTYPE BASE
///RECTAN
///RCONF 0,0,0,0,0,0,0,0,0,0,0,0,0,0,0,0,0,0,0,0,0,0,0,0
P00006=0.222,-3.123,-1.508,0.0000,0.0000,0.0000
P00021=-0.225,-6.128,-0.405,0.0000,0.0000,0.0000
P00022=0.222,-3.123,-1.508,0.0000,0.0000,0.0000
P00023=0.143,-0.036,0.682,0.0000,0.0000,0.0000
P00024=0.145,-0.552,1.326,0.0000,0.0000,0.0000
P00025=-2.003,0.006,0.728,0.0000,0.0000,0.0000
P00026=0.562,-0.002,-0.337,0.0000,0.0000,0.0000
P00027=-0.746,0.015,-9.096,0.0000,0.0000,0.0000
P00028=-2.237,-0.018,-7.702,0.0000,0.0000,0.0000
P00029=-2.156,-0.086,-4.681,0.0000,0.0000,0.0000
P00030=5.926,-4.294,-1.390,0.0000,0.0000,0.0000
P00031=1.853,-0.001,-1.549,0.0000,0.0000,0.0000
P00032=1.957,0.503,-7.217,0.0000,0.0000,0.0000
///RCONF 0,0,0,0,1,0,0,0,0,0,0,0,0,0,0,0,0,0,0,0,0,0,0,0
P00033=-0.123,0.612,-5.012,0.0000,0.0000,0.0000
///RCONF 0,0,0,0,0,0,0,0,0,0,0,0,0,0,0,0,0,0,0,0,0,0,0,0
P00041=0.192,3.924,0.305,0.0000,0.0000,0.0000
P00042=-0.217,1.941,0.413,0.0000,0.0000,0.0000
P00043=-0.044,-1.937,1.197,0.0000,0.0000,0.0000
P00044=0.687,-2.322,1.156,0.0000,0.0000,0.0000
P00045=-0.068,-0.810,1.603,0.0000,0.0000,0.0000
P00046=0.799,0.043,1.292,0.0000,0.0000,0.0000
///RCONF 0,1,0,0,0,0,0,0,0,0,0,0,0,0,0,0,0,0,0,0,0,0,0,0
P00047=-0.011,1.737,-0.646,0.0000,0.0000,0.0000
///RCONF 0,0,0,0,0,0,0,0,0,0,0,0,0,0,0,0,0,0,0,0,0,0,0,0
P00048=2.411,0.025,-0.606,0.0000,0.0000,0.0000
P00049=3.413,-3.572,-1.618,0.0000,0.0000,0.0000
P00050=4.296,-4.501,-0.826,0.0000,0.0000,0.0000
P00051=0.367,3.892,0.009,0.0000,0.0000,0.0000
P00052=0.088,2.832,-0.342,0.0000,0.0000,0.0000
P00053=0.134,6.594,0.107,0.0000,0.0000,0.0000
//INST
///DATE 2024/11/05 11:35
///ATTR SC,RW
///GROUP1 RB1,BS1
///GROUP2 ST1
NOP
'X2_100(P)(125,-90)
'
MOVJ C00000 BC00000 VJ=100.00  +MOVJ EC00000 VJ=100.00
MOVJ C00001 BC00001 VJ=100.00  +MOVJ EC00001 VJ=100.00
'
MOVJ C00002 BC00002 VJ=100.00  +MOVJ EC00002 VJ=100.00
MOVJ C00003 BC00003 VJ=100.00  +MOVJ EC00003 VJ=100.00
MOVJ C00004 BC00004 VJ=100.00  +MOVJ EC00004 VJ=100.00
MOVJ C00005 BC00005 VJ=100.00  +MOVJ EC00005 VJ=100.00
MOVJ C00006 BC00006 VJ=100.00  +MOVJ EC00006 VJ=100.00
'Path S3336
SFTOF3D
MOVJ C00007 BC00007 VJ=100.00  +MOVJ EC00007 VJ=100.00
MOVL C00008 BC00008 V=800.0  +MOVJ EC00008 VJ=100.00
SMOVL C00009 BC00009 V=166.7  +MOVJ EC00009
SREFP 3 C00010 BC00010  +REFP EC00010
CALL JOB:SEARCH-R1-S13D
SET P021 P006
SFTON3D P021
SMOVL C00011 BC00011 V=166.7  +MOVJ EC00011
SREFP 3 C00012 BC00012  +REFP EC00012
CALL JOB:SEARCH-R1-S13D
SET P021 P006
SFTON3D P021
SMOVL C00013 BC00013 V=166.7  +MOVJ EC00013
MOVL C00014 BC00014 V=1000.0  +MOVJ EC00014 VJ=100.00
'EndPath S3336
'Path S3337
SFTOF3D
MOVJ C00015 BC00015 VJ=100.00  +MOVJ EC00015 VJ=100.00
MOVL C00016 BC00016 V=800.0  +MOVJ EC00016 VJ=100.00
SMOVL C00017 BC00017 V=166.7  +MOVJ EC00017
SREFP 3 C00018 BC00018  +REFP EC00018
CALL JOB:SEARCH-R1-S13D
SET P022 P006
SFTON3D P022
SMOVL C00019 BC00019 V=166.7  +MOVJ EC00019
SREFP 3 C00020 BC00020  +REFP EC00020
CALL JOB:SEARCH-R1-S13D
SET P022 P006
SFTON3D P022
SMOVL C00021 BC00021 V=166.7  +MOVJ EC00021
MOVL C00022 BC00022 V=1000.0  +MOVJ EC00022 VJ=100.00
'EndPath S3337
'Path S3338
SFTOF3D
MOVJ C00023 BC00023 VJ=100.00  +MOVJ EC00023 VJ=100.00
MOVL C00024 BC00024 V=800.0  +MOVJ EC00024 VJ=100.00
SMOVL C00025 BC00025 V=166.7  +MOVJ EC00025
SREFP 3 C00026 BC00026  +REFP EC00026
CALL JOB:SEARCH-R1-S13D
SET P023 P006
SFTON3D P023
SMOVL C00027 BC00027 V=166.7  +MOVJ EC00027
SREFP 3 C00028 BC00028  +REFP EC00028
CALL JOB:SEARCH-R1-S13D
SET P023 P006
SFTON3D P023
SMOVL C00029 BC00029 V=166.7  +MOVJ EC00029
MOVL C00030 BC00030 V=1000.0  +MOVJ EC00030 VJ=100.00
'EndPath S3338
MOVJ C00031 BC00031 VJ=100.00  +MOVJ EC00031 VJ=100.00
'Path S3339
SFTOF3D
MOVJ C00032 BC00032 VJ=100.00  +MOVJ EC00032 VJ=100.00
MOVL C00033 BC00033 V=800.0  +MOVJ EC00033 VJ=100.00
SMOVL C00034 BC00034 V=166.7  +MOVJ EC00034
SREFP 3 C00035 BC00035  +REFP EC00035
CALL JOB:SEARCH-R1-S13D
SET P024 P006
SFTON3D P024
SMOVL C00036 BC00036 V=166.7  +MOVJ EC00036
SREFP 3 C00037 BC00037  +REFP EC00037
CALL JOB:SEARCH-R1-S13D
SET P024 P006
SFTON3D P024
SMOVL C00038 BC00038 V=166.7  +MOVJ EC00038
MOVL C00039 BC00039 V=1000.0  +MOVJ EC00039 VJ=100.00
'EndPath S3339
'Path S3341
SFTOF3D
MOVJ C00040 BC00040 VJ=100.00  +MOVJ EC00040 VJ=100.00
MOVL C00041 BC00041 V=800.0  +MOVJ EC00041 VJ=100.00
SMOVL C00042 BC00042 V=166.7  +MOVJ EC00042
SREFP 3 C00043 BC00043  +REFP EC00043
CALL JOB:SEARCH-R1-S13D
SET P025 P006
SFTON3D P025
SMOVL C00044 BC00044 V=166.7  +MOVJ EC00044
SREFP 3 C00045 BC00045  +REFP EC00045
CALL JOB:SEARCH-R1-S13D
SET P025 P006
SFTON3D P025
SMOVL C00046 BC00046 V=166.7  +MOVJ EC00046
MOVL C00047 BC00047 V=1000.0  +MOVJ EC00047 VJ=100.00
'EndPath S3341
'Path S3343
SFTOF3D
MOVJ C00048 BC00048 VJ=100.00  +MOVJ EC00048 VJ=100.00
MOVL C00049 BC00049 V=800.0  +MOVJ EC00049 VJ=100.00
SMOVL C00050 BC00050 V=166.7  +MOVJ EC00050
SREFP 3 C00051 BC00051  +REFP EC00051
CALL JOB:SEARCH-R1-S13D
SET P026 P006
SFTON3D P026
SMOVL C00052 BC00052 V=166.7  +MOVJ EC00052
SREFP 3 C00053 BC00053  +REFP EC00053
CALL JOB:SEARCH-R1-S13D
SET P026 P006
SFTON3D P026
SMOVL C00054 BC00054 V=166.7  +MOVJ EC00054
MOVL C00055 BC00055 V=1000.0  +MOVJ EC00055 VJ=100.00
'EndPath S3343
MOVJ C00056 BC00056 VJ=100.00  +MOVJ EC00056 VJ=100.00
'Path S3345
SFTOF3D
MOVJ C00057 BC00057 VJ=100.00  +MOVJ EC00057 VJ=100.00
MOVL C00058 BC00058 V=800.0  +MOVJ EC00058 VJ=100.00
SMOVL C00059 BC00059 V=166.7  +MOVJ EC00059
SREFP 3 C00060 BC00060  +REFP EC00060
CALL JOB:SEARCH-R1-S13D
SET P027 P006
SFTON3D P027
SMOVL C00061 BC00061 V=166.7  +MOVJ EC00061
SREFP 3 C00062 BC00062  +REFP EC00062
CALL JOB:SEARCH-R1-S13D
SET P027 P006
SFTON3D P027
SMOVL C00063 BC00063 V=166.7  +MOVJ EC00063
MOVL C00064 BC00064 V=1000.0  +MOVJ EC00064 VJ=100.00
'EndPath S3345
MOVJ C00065 BC00065 VJ=100.00  +MOVJ EC00065 VJ=100.00
'Path S3347
SFTOF3D
MOVJ C00066 BC00066 VJ=100.00  +MOVJ EC00066 VJ=100.00
MOVL C00067 BC00067 V=800.0  +MOVJ EC00067 VJ=100.00
SMOVL C00068 BC00068 V=166.7  +MOVJ EC00068
SREFP 3 C00069 BC00069  +REFP EC00069
CALL JOB:SEARCH-R1-S13D
SET P028 P006
SFTON3D P028
SMOVL C00070 BC00070 V=166.7  +MOVJ EC00070
SREFP 3 C00071 BC00071  +REFP EC00071
CALL JOB:SEARCH-R1-S13D
SET P028 P006
SFTON3D P028
SMOVL C00072 BC00072 V=166.7  +MOVJ EC00072
MOVL C00073 BC00073 V=1000.0  +MOVJ EC00073 VJ=100.00
'EndPath S3347
'Path S3349
SFTOF3D
MOVJ C00074 BC00074 VJ=100.00  +MOVJ EC00074 VJ=100.00
MOVL C00075 BC00075 V=800.0  +MOVJ EC00075 VJ=100.00
SMOVL C00076 BC00076 V=166.7  +MOVJ EC00076
SREFP 3 C00077 BC00077  +REFP EC00077
CALL JOB:SEARCH-R1-S13D
SET P029 P006
SFTON3D P029
SMOVL C00078 BC00078 V=166.7  +MOVJ EC00078
SREFP 3 C00079 BC00079  +REFP EC00079
CALL JOB:SEARCH-R1-S13D
SET P029 P006
SFTON3D P029
SMOVL C00080 BC00080 V=166.7  +MOVJ EC00080
MOVL C00081 BC00081 V=1000.0  +MOVJ EC00081 VJ=100.00
'EndPath S3349
'Path S3350
SFTOF3D
MOVJ C00082 BC00082 VJ=100.00  +MOVJ EC00082 VJ=100.00
MOVL C00083 BC00083 V=800.0  +MOVJ EC00083 VJ=100.00
SMOVL C00084 BC00084 V=166.7  +MOVJ EC00084
SREFP 3 C00085 BC00085  +REFP EC00085
CALL JOB:SEARCH-R1-S13D
SET P030 P006
SFTON3D P030
SMOVL C00086 BC00086 V=166.7  +MOVJ EC00086
SREFP 3 C00087 BC00087  +REFP EC00087
CALL JOB:SEARCH-R1-S13D
SET P030 P006
SFTON3D P030
SMOVL C00088 BC00088 V=166.7  +MOVJ EC00088
SMOVL C00089 BC00089 V=166.7  +MOVJ EC00089
SREFP 3 C00090 BC00090  +REFP EC00090
CALL JOB:SEARCH-R1-S13D
SET P030 P006
SFTON3D P030
SMOVL C00091 BC00091 V=166.7  +MOVJ EC00091
MOVL C00092 BC00092 V=1000.0  +MOVJ EC00092 VJ=100.00
'EndPath S3350
'Path S3351
SFTOF3D
MOVJ C00093 BC00093 VJ=100.00  +MOVJ EC00093 VJ=100.00
MOVL C00094 BC00094 V=800.0  +MOVJ EC00094 VJ=100.00
SMOVL C00095 BC00095 V=166.7  +MOVJ EC00095
SREFP 3 C00096 BC00096  +REFP EC00096
CALL JOB:SEARCH-R1-S13D
SET P031 P006
SFTON3D P031
SMOVL C00097 BC00097 V=166.7  +MOVJ EC00097
SREFP 3 C00098 BC00098  +REFP EC00098
CALL JOB:SEARCH-R1-S13D
SET P031 P006
SFTON3D P031
SMOVL C00099 BC00099 V=166.7  +MOVJ EC00099
MOVL C00100 BC00100 V=1000.0  +MOVJ EC00100 VJ=100.00
'EndPath S3351
MOVJ C00101 BC00101 VJ=100.00  +MOVJ EC00101 VJ=100.00
'Path S3352
SFTOF3D
MOVJ C00102 BC00102 VJ=100.00  +MOVJ EC00102 VJ=100.00
MOVL C00103 BC00103 V=800.0  +MOVJ EC00103 VJ=100.00
SMOVL C00104 BC00104 V=166.7  +MOVJ EC00104
SREFP 3 C00105 BC00105  +REFP EC00105
CALL JOB:SEARCH-R1-S13D
SET P032 P006
SFTON3D P032
SMOVL C00106 BC00106 V=166.7  +MOVJ EC00106
SREFP 3 C00107 BC00107  +REFP EC00107
CALL JOB:SEARCH-R1-S13D
SET P032 P006
SFTON3D P032
SMOVL C00108 BC00108 V=166.7  +MOVJ EC00108
MOVL C00109 BC00109 V=1000.0  +MOVJ EC00109 VJ=100.00
'EndPath S3352
'Path S3353
SFTOF3D
MOVJ C00110 BC00110 VJ=100.00  +MOVJ EC00110 VJ=100.00
MOVL C00111 BC00111 V=800.0  +MOVJ EC00111 VJ=100.00
SMOVL C00112 BC00112 V=166.7  +MOVJ EC00112
SREFP 3 C00113 BC00113  +REFP EC00113
CALL JOB:SEARCH-R1-S13D
SET P033 P006
SFTON3D P033
SMOVL C00114 BC00114 V=166.7  +MOVJ EC00114
SREFP 3 C00115 BC00115  +REFP EC00115
CALL JOB:SEARCH-R1-S13D
SET P033 P006
SFTON3D P033
SMOVL C00116 BC00116 V=166.7  +MOVJ EC00116
MOVL C00117 BC00117 V=1000.0  +MOVJ EC00117 VJ=100.00
'EndPath S3353
MOVJ C00118 BC00118 VJ=100.00  +MOVJ EC00118 VJ=100.00
MOVJ C00119 BC00119 VJ=100.00  +MOVJ EC00119 VJ=100.00
'Path W3292
SFTOF3D
SFTON3D P021
MOVJ C00120 BC00120 VJ=100.00  +MOVJ EC00120 VJ=100.00
SMOVL C00121 BC00121 V=800.0  +MOVJ EC00121
SMOVL C00122 BC00122 V=166.7 PL=0  +MOVJ EC00122
MACRO1 MJ#(0) ARGF9
ARCON
SMOVL C00123 BC00123 V=11.7  +MOVJ EC00123
SMOVL C00124 BC00124 V=11.7  +MOVJ EC00124
SMOVL C00125 BC00125 V=11.7  +MOVJ EC00125
ARCOF
SMOVL C00126 BC00126 V=800.0  +MOVJ EC00126
SMOVL C00127 BC00127 V=1000.0  +MOVJ EC00127
SFTOF3D
'EndPath W3292
'Path W3293
SFTOF3D
SFTON3D P022
MOVJ C00128 BC00128 VJ=100.00  +MOVJ EC00128 VJ=100.00
SMOVL C00129 BC00129 V=800.0  +MOVJ EC00129
SMOVL C00130 BC00130 V=166.7 PL=0  +MOVJ EC00130
ARCON
SMOVL C00131 BC00131 V=11.7  +MOVJ EC00131
ARCOF
SMOVL C00132 BC00132 V=800.0  +MOVJ EC00132
SMOVL C00133 BC00133 V=1000.0  +MOVJ EC00133
SFTOF3D
'EndPath W3293
'Path W3294
SFTOF3D
SFTON3D P023
MOVJ C00134 BC00134 VJ=100.00  +MOVJ EC00134 VJ=100.00
SMOVL C00135 BC00135 V=800.0  +MOVJ EC00135
SMOVL C00136 BC00136 V=166.7 PL=0  +MOVJ EC00136
ARCON
SMOVL C00137 BC00137 V=11.7  +MOVJ EC00137
ARCOF
SMOVL C00138 BC00138 V=800.0  +MOVJ EC00138
SMOVL C00139 BC00139 V=1000.0  +MOVJ EC00139
SFTOF3D
'EndPath W3294
'
MOVJ C00140 BC00140 VJ=100.00  +MOVJ EC00140 VJ=100.00
'Path W3340
SFTOF3D
SFTON3D P024
MOVJ C00141 BC00141 VJ=100.00  +MOVJ EC00141 VJ=100.00
SMOVL C00142 BC00142 V=800.0  +MOVJ EC00142
SMOVL C00143 BC00143 V=150.0 PL=0  +MOVJ EC00143
ARCON
SMOVL C00144 BC00144 V=11.7  +MOVJ EC00144
SMOVL C00145 BC00145 V=11.7  +MOVJ EC00145
SMOVL C00146 BC00146 V=11.7  +MOVJ EC00146
ARCOF
SMOVL C00147 BC00147 V=800.0  +MOVJ EC00147
SMOVL C00148 BC00148 V=1000.0  +MOVJ EC00148
SFTOF3D
'EndPath W3340
'Path W3342
SFTOF3D
SFTON3D P025
MOVJ C00149 BC00149 VJ=100.00  +MOVJ EC00149 VJ=100.00
SMOVL C00150 BC00150 V=800.0  +MOVJ EC00150
SMOVL C00151 BC00151 V=150.0 PL=0  +MOVJ EC00151
ARCON
SMOVL C00152 BC00152 V=11.7  +MOVJ EC00152
ARCOF
SMOVL C00153 BC00153 V=800.0  +MOVJ EC00153
SMOVL C00154 BC00154 V=1000.0  +MOVJ EC00154
SFTOF3D
'EndPath W3342
'Path W3344
SFTOF3D
SFTON3D P026
MOVJ C00155 BC00155 VJ=100.00  +MOVJ EC00155 VJ=100.00
SMOVL C00156 BC00156 V=800.0  +MOVJ EC00156
SMOVL C00157 BC00157 V=150.0 PL=0  +MOVJ EC00157
ARCON
SMOVL C00158 BC00158 V=11.7  +MOVJ EC00158
ARCOF
SMOVL C00159 BC00159 V=800.0  +MOVJ EC00159
SMOVL C00160 BC00160 V=1000.0  +MOVJ EC00160
SFTOF3D
'EndPath W3344
'
MOVJ C00161 BC00161 VJ=100.00  +MOVJ EC00161 VJ=100.00
'Path W3346
SFTOF3D
SFTON3D P027
MOVJ C00162 BC00162 VJ=100.00  +MOVJ EC00162 VJ=100.00
SMOVL C00163 BC00163 V=800.0  +MOVJ EC00163
SMOVL C00164 BC00164 V=150.0 PL=0  +MOVJ EC00164
ARCON
SMOVL C00165 BC00165 V=11.7  +MOVJ EC00165
ARCOF
SMOVL C00166 BC00166 V=800.0  +MOVJ EC00166
SMOVL C00167 BC00167 V=1000.0  +MOVJ EC00167
SFTOF3D
'EndPath W3346
'Path W3348
SFTOF3D
SFTON3D P028
MOVJ C00168 BC00168 VJ=100.00  +MOVJ EC00168 VJ=100.00
SMOVL C00169 BC00169 V=800.0  +MOVJ EC00169
SMOVL C00170 BC00170 V=150.0 PL=0  +MOVJ EC00170
ARCON
SMOVL C00171 BC00171 V=11.7  +MOVJ EC00171
ARCOF
SMOVL C00172 BC00172 V=800.0  +MOVJ EC00172
SMOVL C00173 BC00173 V=1000.0  +MOVJ EC00173
SFTOF3D
'EndPath W3348
'Path W3350
SFTOF3D
SFTON3D P029
MOVJ C00174 BC00174 VJ=100.00  +MOVJ EC00174 VJ=100.00
SMOVL C00175 BC00175 V=800.0  +MOVJ EC00175
SMOVL C00176 BC00176 V=150.0 PL=0  +MOVJ EC00176
ARCON
SMOVL C00177 BC00177 V=11.7  +MOVJ EC00177
SMOVL C00178 BC00178 V=11.7  +MOVJ EC00178
ARCOF
SMOVL C00179 BC00179 V=800.0  +MOVJ EC00179
SMOVL C00180 BC00180 V=1000.0  +MOVJ EC00180
SFTOF3D
'EndPath W3350
MOVJ C00181 BC00181 VJ=100.00  +MOVJ EC00181 VJ=100.00
'
'Path W3316
SFTOF3D
SFTON3D P031
MOVJ C00182 BC00182 VJ=100.00  +MOVJ EC00182 VJ=100.00
SMOVL C00183 BC00183 V=800.0  +MOVJ EC00183
SMOVL C00184 BC00184 V=150.0 PL=0  +MOVJ EC00184
MACRO1 MJ#(0) ARGF21
ARCON
SMOVL C00185 BC00185 V=10.0  +MOVJ EC00185
SFTON3D P030
SMOVL C00186 BC00186 V=10.0  +MOVJ EC00186
SMOVL C00187 BC00187 V=10.0  +MOVJ EC00187
ARCOF
SMOVL C00188 BC00188 V=800.0  +MOVJ EC00188
SMOVL C00189 BC00189 V=1000.0  +MOVJ EC00189
SFTOF3D
'EndPath W3316
MOVJ C00190 BC00190 VJ=100.00  +MOVJ EC00190 VJ=100.00
'
'Path W3319
SFTOF3D
SFTON3D P032
MOVJ C00191 BC00191 VJ=100.00  +MOVJ EC00191 VJ=100.00
SMOVL C00192 BC00192 V=800.0  +MOVJ EC00192
SMOVL C00193 BC00193 V=150.0 PL=0  +MOVJ EC00193
ARCON
SFTON3D P033
SMOVL C00194 BC00194 V=9.2  +MOVJ EC00194
ARCOF
SMOVL C00195 BC00195 V=800.0  +MOVJ EC00195
SMOVL C00196 BC00196 V=1000.0  +MOVJ EC00196
SFTOF3D
'EndPath W3319
MOVJ C00197 BC00197 VJ=100.00  +MOVJ EC00197 VJ=100.00
MOVJ C00198 BC00198 VJ=100.00  +MOVJ EC00198 VJ=100.00
'
MOVJ C00199 BC00199 VJ=100.00  +MOVJ EC00199 VJ=100.00
MOVJ C00200 BC00200 VJ=100.00  +MOVJ EC00200 VJ=100.00
CALL JOB:CLEAN-R1_KM_NEW
'CUT-WIRE !!!!
MOVJ C00201 BC00201 VJ=100.00  +MOVJ EC00201 VJ=100.00
MOVJ C00202 BC00202 VJ=100.00  +MOVJ EC00202 VJ=100.00
MOVJ C00203 BC00203 VJ=100.00  +MOVJ EC00203 VJ=100.00
MOVJ C00204 BC00204 VJ=100.00  +MOVJ EC00204 VJ=100.00
MOVJ C00205 BC00205 VJ=100.00  +MOVJ EC00205 VJ=100.00
'
'Path S3355
SFTOF3D
MOVJ C00206 BC00206 VJ=100.00  +MOVJ EC00206 VJ=100.00
MOVL C00207 BC00207 V=800.0  +MOVJ EC00207 VJ=100.00
MOVL C00208 BC00208 V=800.0  +MOVJ EC00208 VJ=100.00
SMOVL C00209 BC00209 V=166.7  +MOVJ EC00209
SREFP 3 C00210 BC00210  +REFP EC00210
CALL JOB:SEARCH-R1-S13D
SET P041 P006
SFTON3D P041
SMOVL C00211 BC00211 V=166.7  +MOVJ EC00211
SREFP 3 C00212 BC00212  +REFP EC00212
CALL JOB:SEARCH-R1-S13D
SET P041 P006
SFTON3D P041
SMOVL C00213 BC00213 V=166.7  +MOVJ EC00213
MOVL C00214 BC00214 V=1000.0  +MOVJ EC00214 VJ=100.00
'EndPath S3355
'Path S3356
SFTOF3D
MOVJ C00215 BC00215 VJ=100.00  +MOVJ EC00215 VJ=100.00
MOVL C00216 BC00216 V=800.0  +MOVJ EC00216 VJ=100.00
SMOVL C00217 BC00217 V=166.7  +MOVJ EC00217
SREFP 3 C00218 BC00218  +REFP EC00218
CALL JOB:SEARCH-R1-S13D
SET P042 P006
SFTON3D P042
SMOVL C00219 BC00219 V=166.7  +MOVJ EC00219
SREFP 3 C00220 BC00220  +REFP EC00220
CALL JOB:SEARCH-R1-S13D
SET P042 P006
SFTON3D P042
SMOVL C00221 BC00221 V=166.7  +MOVJ EC00221
MOVL C00222 BC00222 V=1000.0  +MOVJ EC00222 VJ=100.00
'EndPath S3356
MOVJ C00223 BC00223 VJ=100.00  +MOVJ EC00223 VJ=100.00
MOVJ C00224 BC00224 VJ=100.00  +MOVJ EC00224 VJ=100.00
'Path S3357
SFTOF3D
MOVJ C00225 BC00225 VJ=100.00  +MOVJ EC00225 VJ=100.00
MOVL C00226 BC00226 V=800.0  +MOVJ EC00226 VJ=100.00
SMOVL C00227 BC00227 V=166.7  +MOVJ EC00227
SREFP 3 C00228 BC00228  +REFP EC00228
CALL JOB:SEARCH-R1-S13D
SET P043 P006
SFTON3D P043
SMOVL C00229 BC00229 V=166.7  +MOVJ EC00229
SREFP 3 C00230 BC00230  +REFP EC00230
CALL JOB:SEARCH-R1-S13D
SET P043 P006
SFTON3D P043
MOVL C00231 BC00231 V=800.0  +MOVJ EC00231 VJ=100.00
MOVL C00232 BC00232 V=500.0  +MOVJ EC00232 VJ=100.00
'EndPath S3357
MOVJ C00233 BC00233 VJ=100.00  +MOVJ EC00233 VJ=100.00
'Path S3358
SFTOF3D
MOVJ C00234 BC00234 VJ=100.00  +MOVJ EC00234 VJ=100.00
MOVL C00235 BC00235 V=800.0  +MOVJ EC00235 VJ=100.00
SMOVL C00236 BC00236 V=166.7  +MOVJ EC00236
SREFP 3 C00237 BC00237  +REFP EC00237
CALL JOB:SEARCH-R1-S13D
SET P044 P006
SFTON3D P044
SMOVL C00238 BC00238 V=166.7  +MOVJ EC00238
SREFP 3 C00239 BC00239  +REFP EC00239
CALL JOB:SEARCH-R1-S13D
SET P044 P006
SFTON3D P044
SMOVL C00240 BC00240 V=166.7  +MOVJ EC00240
MOVL C00241 BC00241 V=1000.0  +MOVJ EC00241 VJ=100.00
'EndPath S3358
'Path S3359
SFTOF3D
MOVJ C00242 BC00242 VJ=100.00  +MOVJ EC00242 VJ=100.00
MOVL C00243 BC00243 V=800.0  +MOVJ EC00243 VJ=100.00
SMOVL C00244 BC00244 V=166.7  +MOVJ EC00244
SREFP 3 C00245 BC00245  +REFP EC00245
CALL JOB:SEARCH-R1-S13D
SET P045 P006
SFTON3D P045
SMOVL C00246 BC00246 V=166.7  +MOVJ EC00246
SREFP 3 C00247 BC00247  +REFP EC00247
CALL JOB:SEARCH-R1-S13D
SET P045 P006
SFTON3D P045
SMOVL C00248 BC00248 V=166.7  +MOVJ EC00248
MOVL C00249 BC00249 V=1000.0  +MOVJ EC00249 VJ=100.00
'EndPath S3359
'Path S3360
SFTOF3D
MOVJ C00250 BC00250 VJ=100.00  +MOVJ EC00250 VJ=100.00
MOVL C00251 BC00251 V=800.0  +MOVJ EC00251 VJ=100.00
SMOVL C00252 BC00252 V=166.7  +MOVJ EC00252
SREFP 3 C00253 BC00253  +REFP EC00253
CALL JOB:SEARCH-R1-S13D
SET P046 P006
SFTON3D P046
SMOVL C00254 BC00254 V=166.7  +MOVJ EC00254
SREFP 3 C00255 BC00255  +REFP EC00255
CALL JOB:SEARCH-R1-S13D
SET P046 P006
SFTON3D P046
SMOVL C00256 BC00256 V=166.7  +MOVJ EC00256
MOVL C00257 BC00257 V=1000.0  +MOVJ EC00257 VJ=100.00
'EndPath S3360
MOVJ C00258 BC00258 VJ=100.00  +MOVJ EC00258 VJ=100.00
'Path S3361
SFTOF3D
MOVJ C00259 BC00259 VJ=100.00  +MOVJ EC00259 VJ=100.00
MOVL C00260 BC00260 V=800.0  +MOVJ EC00260 VJ=100.00
SMOVL C00261 BC00261 V=166.7  +MOVJ EC00261
SREFP 3 C00262 BC00262  +REFP EC00262
CALL JOB:SEARCH-R1-S13D
SET P047 P006
SFTON3D P047
SMOVL C00263 BC00263 V=166.7  +MOVJ EC00263
SREFP 3 C00264 BC00264  +REFP EC00264
CALL JOB:SEARCH-R1-S13D
SET P047 P006
SFTON3D P047
SMOVL C00265 BC00265 V=166.7  +MOVJ EC00265
MOVL C00266 BC00266 V=1000.0  +MOVJ EC00266 VJ=100.00
'EndPath S3361
'Path S3362
SFTOF3D
MOVJ C00267 BC00267 VJ=100.00  +MOVJ EC00267 VJ=100.00
MOVL C00268 BC00268 V=800.0  +MOVJ EC00268 VJ=100.00
SMOVL C00269 BC00269 V=166.7  +MOVJ EC00269
SREFP 3 C00270 BC00270  +REFP EC00270
CALL JOB:SEARCH-R1-S13D
SET P048 P006
SFTON3D P048
SMOVL C00271 BC00271 V=166.7  +MOVJ EC00271
SREFP 3 C00272 BC00272  +REFP EC00272
CALL JOB:SEARCH-R1-S13D
SET P048 P006
SFTON3D P048
SMOVL C00273 BC00273 V=166.7  +MOVJ EC00273
MOVL C00274 BC00274 V=1000.0  +MOVJ EC00274 VJ=100.00
'EndPath S3362
'Path S3363
SFTOF3D
MOVJ C00275 BC00275 VJ=100.00  +MOVJ EC00275 VJ=100.00
MOVL C00276 BC00276 V=800.0  +MOVJ EC00276 VJ=100.00
SMOVL C00277 BC00277 V=166.7  +MOVJ EC00277
SREFP 3 C00278 BC00278  +REFP EC00278
CALL JOB:SEARCH-R1-S13D
SET P049 P006
SFTON3D P049
SMOVL C00279 BC00279 V=166.7  +MOVJ EC00279
SREFP 3 C00280 BC00280  +REFP EC00280
CALL JOB:SEARCH-R1-S13D
SET P049 P006
SFTON3D P049
SMOVL C00281 BC00281 V=166.7  +MOVJ EC00281
MOVL C00282 BC00282 V=1000.0  +MOVJ EC00282 VJ=100.00
'EndPath S3363
'Path S3364
SFTOF3D
MOVJ C00283 BC00283 VJ=100.00  +MOVJ EC00283 VJ=100.00
MOVJ C00284 BC00284 VJ=100.00  +MOVJ EC00284 VJ=100.00
MOVL C00285 BC00285 V=800.0  +MOVJ EC00285 VJ=100.00
SMOVL C00286 BC00286 V=166.7  +MOVJ EC00286
SREFP 3 C00287 BC00287  +REFP EC00287
CALL JOB:SEARCH-R1-S13D
SET P050 P006
SFTON3D P050
SMOVL C00288 BC00288 V=166.7  +MOVJ EC00288
SREFP 3 C00289 BC00289  +REFP EC00289
CALL JOB:SEARCH-R1-S13D
SET P050 P006
SFTON3D P050
SMOVL C00290 BC00290 V=166.7  +MOVJ EC00290
'EndPath S3364
'Path S3365
SFTOF3D
MOVJ C00291 BC00291 VJ=100.00  +MOVJ EC00291 VJ=100.00
MOVL C00292 BC00292 V=800.0  +MOVJ EC00292 VJ=100.00
SMOVL C00293 BC00293 V=166.7  +MOVJ EC00293
SREFP 3 C00294 BC00294  +REFP EC00294
CALL JOB:SEARCH-R1-S13D
SET P051 P006
SFTON3D P051
SMOVL C00295 BC00295 V=166.7  +MOVJ EC00295
SREFP 3 C00296 BC00296  +REFP EC00296
CALL JOB:SEARCH-R1-S13D
SET P051 P006
SFTON3D P051
SMOVL C00297 BC00297 V=166.7  +MOVJ EC00297
MOVL C00298 BC00298 V=1000.0  +MOVJ EC00298 VJ=100.00
'EndPath S3365
MOVJ C00299 BC00299 VJ=100.00  +MOVJ EC00299 VJ=100.00
'Path S3366
SFTOF3D
MOVJ C00300 BC00300 VJ=100.00  +MOVJ EC00300 VJ=100.00
MOVL C00301 BC00301 V=800.0  +MOVJ EC00301 VJ=100.00
SMOVL C00302 BC00302 V=166.7  +MOVJ EC00302
SREFP 3 C00303 BC00303  +REFP EC00303
CALL JOB:SEARCH-R1-S13D
SET P052 P006
SFTON3D P052
SMOVL C00304 BC00304 V=166.7  +MOVJ EC00304
SREFP 3 C00305 BC00305  +REFP EC00305
CALL JOB:SEARCH-R1-S13D
SET P052 P006
SFTON3D P052
SMOVL C00306 BC00306 V=166.7  +MOVJ EC00306
MOVL C00307 BC00307 V=1000.0  +MOVJ EC00307 VJ=100.00
'EndPath S3366
'Path S3367
SFTOF3D
MOVJ C00308 BC00308 VJ=100.00  +MOVJ EC00308 VJ=100.00
MOVL C00309 BC00309 V=800.0  +MOVJ EC00309 VJ=100.00
SMOVL C00310 BC00310 V=166.7  +MOVJ EC00310
SREFP 3 C00311 BC00311  +REFP EC00311
CALL JOB:SEARCH-R1-S13D
SET P053 P006
SFTON3D P053
SMOVL C00312 BC00312 V=166.7  +MOVJ EC00312
SREFP 3 C00313 BC00313  +REFP EC00313
CALL JOB:SEARCH-R1-S13D
SET P053 P006
SFTON3D P053
SMOVL C00314 BC00314 V=166.7  +MOVJ EC00314
SFTOF3D
MOVL C00315 BC00315 V=1000.0  +MOVJ EC00315 VJ=100.00
'EndPath S3367
'
'Path W3331
SFTOF3D
SFTON3D P052
MOVJ C00316 BC00316 VJ=100.00  +MOVJ EC00316 VJ=100.00
SMOVL C00317 BC00317 V=800.0  +MOVJ EC00317
SMOVL C00318 BC00318 V=150.0 PL=0  +MOVJ EC00318
ARCON
SFTON3D P053
SMOVL C00319 BC00319 V=9.2  +MOVJ EC00319
ARCOF
SMOVL C00320 BC00320 V=800.0  +MOVJ EC00320
SMOVL C00321 BC00321 V=1000.0  +MOVJ EC00321
SFTOF3D
'EndPath W3331
MOVJ C00322 BC00322 VJ=100.00  +MOVJ EC00322 VJ=100.00
'
'Path W3335
SFTOF3D
SFTON3D P051
MOVJ C00323 BC00323 VJ=100.00  +MOVJ EC00323 VJ=100.00
SMOVL C00324 BC00324 V=800.0  +MOVJ EC00324
SMOVL C00325 BC00325 V=150.0 PL=0  +MOVJ EC00325
ARCON
SFTON3D P050
SMOVL C00326 BC00326 V=9.2  +MOVJ EC00326
ARCOF
SMOVL C00327 BC00327 V=800.0  +MOVJ EC00327
SMOVL C00328 BC00328 V=1000.0  +MOVJ EC00328
SFTOF3D
'EndPath W3335
'
'Path W3326
SFTOF3D
SFTON3D P047
MOVJ C00329 BC00329 VJ=100.00  +MOVJ EC00329 VJ=100.00
SMOVL C00330 BC00330 V=800.0  +MOVJ EC00330
SMOVL C00331 BC00331 V=150.0 PL=0  +MOVJ EC00331
MACRO1 MJ#(0) ARGF9
ARCON
SMOVL C00332 BC00332 V=11.7  +MOVJ EC00332
ARCOF
SMOVL C00333 BC00333 V=800.0  +MOVJ EC00333
SMOVL C00334 BC00334 V=1000.0  +MOVJ EC00334
SFTOF3D
'EndPath W3326
'Path W3327
SFTOF3D
SFTON3D P048
MOVJ C00335 BC00335 VJ=100.00  +MOVJ EC00335 VJ=100.00
SMOVL C00336 BC00336 V=800.0  +MOVJ EC00336
SMOVL C00337 BC00337 V=150.0 PL=0  +MOVJ EC00337
ARCON
SMOVL C00338 BC00338 V=11.7  +MOVJ EC00338
ARCOF
SMOVL C00339 BC00339 V=800.0  +MOVJ EC00339
SMOVL C00340 BC00340 V=1000.0  +MOVJ EC00340
SFTOF3D
'EndPath W3327
'Path W3328
SFTOF3D
SFTON3D P049
MOVJ C00341 BC00341 VJ=100.00  +MOVJ EC00341 VJ=100.00
SMOVL C00342 BC00342 V=800.0  +MOVJ EC00342
SMOVL C00343 BC00343 V=150.0 PL=0  +MOVJ EC00343
ARCON
SMOVL C00344 BC00344 V=11.7  +MOVJ EC00344
SMOVL C00345 BC00345 V=11.7  +MOVJ EC00345
ARCOF
SMOVL C00346 BC00346 V=800.0  +MOVJ EC00346
SMOVL C00347 BC00347 V=1000.0  +MOVJ EC00347
SFTOF3D
'EndPath W3328
MOVJ C00348 BC00348 VJ=100.00  +MOVJ EC00348 VJ=100.00
'
'Path W3323
SFTOF3D
SFTON3D P044
MOVJ C00349 BC00349 VJ=100.00  +MOVJ EC00349 VJ=100.00
SMOVL C00350 BC00350 V=800.0  +MOVJ EC00350
SMOVL C00351 BC00351 V=150.0 PL=0  +MOVJ EC00351
ARCON
SMOVL C00352 BC00352 V=11.7  +MOVJ EC00352
SMOVL C00353 BC00353 V=11.7  +MOVJ EC00353
ARCOF
SMOVL C00354 BC00354 V=800.0  +MOVJ EC00354
SMOVL C00355 BC00355 V=1000.0  +MOVJ EC00355
SFTOF3D
'EndPath W3323
'Path W3324
SFTOF3D
SFTON3D P045
MOVJ C00356 BC00356 VJ=100.00  +MOVJ EC00356 VJ=100.00
SMOVL C00357 BC00357 V=800.0  +MOVJ EC00357
SMOVL C00358 BC00358 V=150.0 PL=0  +MOVJ EC00358
ARCON
SMOVL C00359 BC00359 V=11.7  +MOVJ EC00359
ARCOF
SMOVL C00360 BC00360 V=800.0  +MOVJ EC00360
SMOVL C00361 BC00361 V=1000.0  +MOVJ EC00361
SFTOF3D
'EndPath W3324
'Path W3325
SFTOF3D
SFTON3D P046
MOVJ C00362 BC00362 VJ=100.00  +MOVJ EC00362 VJ=100.00
SMOVL C00363 BC00363 V=800.0  +MOVJ EC00363
SMOVL C00364 BC00364 V=150.0 PL=0  +MOVJ EC00364
ARCON
SMOVL C00365 BC00365 V=11.7  +MOVJ EC00365
ARCOF
SMOVL C00366 BC00366 V=800.0  +MOVJ EC00366
SMOVL C00367 BC00367 V=1000.0  +MOVJ EC00367
SFTOF3D
'EndPath W3325
MOVJ C00368 BC00368 VJ=100.00  +MOVJ EC00368 VJ=100.00
'
'
'Path W3320
SFTOF3D
SFTON3D P041
MOVJ C00369 BC00369 VJ=100.00  +MOVJ EC00369 VJ=100.00
SMOVL C00370 BC00370 V=800.0  +MOVJ EC00370
SMOVL C00371 BC00371 V=166.7 PL=0  +MOVJ EC00371
ARCON
SMOVL C00372 BC00372 V=11.7  +MOVJ EC00372
ARCOF
SMOVL C00373 BC00373 V=800.0  +MOVJ EC00373
SMOVL C00374 BC00374 V=1000.0  +MOVJ EC00374
SFTOF3D
'EndPath W3320
'Path W3321
SFTOF3D
SFTON3D P042
MOVJ C00375 BC00375 VJ=100.00  +MOVJ EC00375 VJ=100.00
SMOVL C00376 BC00376 V=800.0  +MOVJ EC00376
SMOVL C00377 BC00377 V=166.7 PL=0  +MOVJ EC00377
ARCON
SMOVL C00378 BC00378 V=11.7  +MOVJ EC00378
ARCOF
SMOVL C00379 BC00379 V=800.0  +MOVJ EC00379
SMOVL C00380 BC00380 V=1000.0  +MOVJ EC00380
SFTOF3D
'EndPath W3321
'Path W3322
SFTOF3D
SFTON3D P043
MOVJ C00381 BC00381 VJ=100.00  +MOVJ EC00381 VJ=100.00
SMOVL C00382 BC00382 V=800.0  +MOVJ EC00382
SMOVL C00383 BC00383 V=166.7 PL=0  +MOVJ EC00383
ARCON
SMOVL C00384 BC00384 V=11.7  +MOVJ EC00384
SMOVL C00385 BC00385 V=11.7  +MOVJ EC00385
ARCOF
SMOVL C00386 BC00386 V=800.0  +MOVJ EC00386
SMOVL C00387 BC00387 V=1000.0  +MOVJ EC00387
SFTOF3D
'EndPath W3322
MOVJ C00388 BC00388 VJ=100.00  +MOVJ EC00388 VJ=100.00
MOVJ C00389 BC00389 VJ=100.00  +MOVJ EC00389 VJ=100.00
MOVJ C00390 BC00390 VJ=100.00  +MOVJ EC00390 VJ=100.00
END
